// TIA Portal V18 export
FUNCTION "RollerV2" : Void   // FC16, LAD
{ S7_Optimized_Access := 'TRUE' }
AUTHOR : HenriP
VERSION : 0.1
// Module behave as a flip flip switch for the Start and Stop Command
// stored: AutoNumber true, IsIECCheckEnabled false, SetENOAutomatically false, UDAEnableTagReadback false
   VAR_INPUT
      SystemON : Bool;
   END_VAR
   VAR_IN_OUT
      Start : Bool;
      Stop : Bool;
      ORoller : Bool;
   END_VAR
BEGIN

REGION Network 1: RollerON
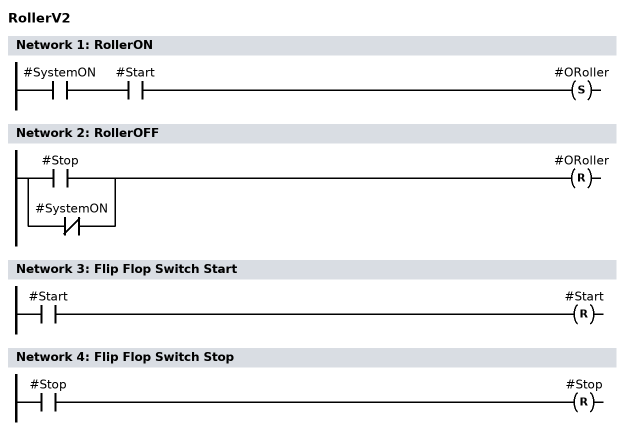
   RUNG wire#powerrail
      Contact( #SystemON )
      Contact( #Start )
      S_Coil( #ORoller )
   END_RUNG
   // the same network as SCL:
   IF #SystemON AND #Start THEN #ORoller := TRUE; END_IF;
END_REGION

REGION Network 2: RollerOFF
   RUNG wire#powerrail
      Contact( #Stop )
      wire#w1
      R_Coil( #ORoller )
   END_RUNG
   RUNG wire#powerrail
      I_Contact( #SystemON )
   END_RUNG wire#w1
   // the same network as SCL:
   IF #Stop OR NOT #SystemON THEN #ORoller := FALSE; END_IF;
END_REGION

REGION Network 3: Flip Flop Switch Start
   RUNG wire#powerrail
      Contact( #Start )
      R_Coil( #Start )
   END_RUNG
   // the same network as SCL:
   IF #Start THEN #Start := FALSE; END_IF;
END_REGION

REGION Network 4: Flip Flop Switch Stop
   RUNG wire#powerrail
      Contact( #Stop )
      R_Coil( #Stop )
   END_RUNG
   // the same network as SCL:
   IF #Stop THEN #Stop := FALSE; END_IF;
END_REGION
END_FUNCTION
